// TIA Portal project "Modbus TCP Example with ESP32" (V16)

(* hardware
DEVICE "S7-1200 station_1"  S7-1200 Station
   slot 0: "Rack_0"  S7-1200 Rack  Rack  V1.0
   slot 1: "PLC_1"  CPU 1211C DC/DC/DC  6ES7 211-1AE40-0XB0  V4.4
*)

// ===== PLC "PLC_1"  CPU 1211C DC/DC/DC =====

VAR_GLOBAL   // PLC tag table "Default tag table"
   "Tag_1" AT %Q0.0 : Bool;
   "System_Byte" AT %MB1 : Byte;
   "FirstScan" AT %M1.0 : Bool;
   "DiagStatusUpdate" AT %M1.1 : Bool;
   "AlwaysTRUE" AT %M1.2 : Bool;
   "AlwaysFALSE" AT %M1.3 : Bool;
   "Clock_Byte" AT %MB0 : Byte;
   "Clock_10Hz" AT %M0.0 : Bool;
   "Clock_5Hz" AT %M0.1 : Bool;
   "Clock_2.5Hz" AT %M0.2 : Bool;
   "Clock_2Hz" AT %M0.3 : Bool;
   "Clock_1.25Hz" AT %M0.4 : Bool;
   "Clock_1Hz" AT %M0.5 : Bool;
   "Clock_0.625Hz" AT %M0.6 : Bool;
   "Clock_0.5Hz" AT %M0.7 : Bool;
END_VAR

TYPE "Modbus TCP FC01-02"
   STRUCT
      REQ : Bool := false;
      DISCONNECT : Bool := false;
      MODE : USInt;
      DATA_ADDR : UDInt;
      DATA_LEN : UInt := 40;
      CONNECT : TCON_IP_v4;
      DONE : Bool := false;
      BUSY : Bool := false;
      ERROR : Bool := false;
      STATUS : Word := 16#0;
      Data : Array[0..39] of Bool;
   END_STRUCT;
   // CONNECT.InterfaceId := 64;
   // CONNECT.ID := 1;
   // CONNECT.ConnectionType := 11;
   // CONNECT.ActiveEstablished := true;
   // CONNECT.RemoteAddress.ADDR[1] := 192;
   // CONNECT.RemoteAddress.ADDR[2] := 168;
   // CONNECT.RemoteAddress.ADDR[3] := 100;
   // CONNECT.RemoteAddress.ADDR[4] := 36;
   // CONNECT.RemotePort := 502;
END_TYPE

TYPE "Modbus TCP FC03-04"
   STRUCT
      REQ : Bool := false;
      DISCONNECT : Bool := false;
      MODE : USInt;
      DATA_ADDR : UDInt;
      DATA_LEN : UInt := 40;
      CONNECT : TCON_IP_v4;
      DONE : Bool := false;
      BUSY : Bool := false;
      ERROR : Bool := false;
      STATUS : Word := 16#0;
      Data : Array[0..39] of UInt;
   END_STRUCT;
   // CONNECT.InterfaceId := 64;
   // CONNECT.ID := 1;
   // CONNECT.ConnectionType := 11;
   // CONNECT.ActiveEstablished := true;
   // CONNECT.RemoteAddress.ADDR[1] := 192;
   // CONNECT.RemoteAddress.ADDR[2] := 168;
   // CONNECT.RemoteAddress.ADDR[3] := 100;
   // CONNECT.RemoteAddress.ADDR[4] := 36;
   // CONNECT.RemotePort := 502;
END_TYPE

DATA_BLOCK "Modbus client"   // DB3
{ S7_Optimized_Access := 'TRUE' }
VERSION : 0.1
   VAR
      Coils : "Modbus TCP FC01-02";
      "Discrete Inputs" : "Modbus TCP FC01-02";
      "Holding Registers" : "Modbus TCP FC03-04";
      "Input Registers" : "Modbus TCP FC03-04";
   END_VAR
BEGIN
   Coils.MODE := 1;
   Coils.DATA_ADDR := 1;
   "Discrete Inputs".MODE := 0;
   "Discrete Inputs".DATA_ADDR := 10101;
   "Discrete Inputs".DATA_LEN := 40;
   Coils.DATA_LEN := 40;
   "Holding Registers".MODE := 1;
   "Holding Registers".DATA_ADDR := 40201;
   "Holding Registers".DATA_LEN := 40;
   "Input Registers".MODE := 0;
   "Input Registers".DATA_ADDR := 30301;
   "Input Registers".DATA_LEN := 40;
END_DATA_BLOCK

ORGANIZATION_BLOCK "Main"   // OB1, LAD, ProgramCycle
TITLE = "Main Program Sweep (Cycle)"
{ S7_Optimized_Access := 'TRUE' }
VERSION : 0.1
   VAR_INPUT
      Initial_Call : Bool;   // Initial call of this OB
      Remanence : Bool;   // =True, if remanent data are available
   END_VAR
   VAR_TEMP
      start : Bool;
      trig1 : Bool;
      trig2 : Bool;
   END_VAR
BEGIN

REGION Network 1: Coils
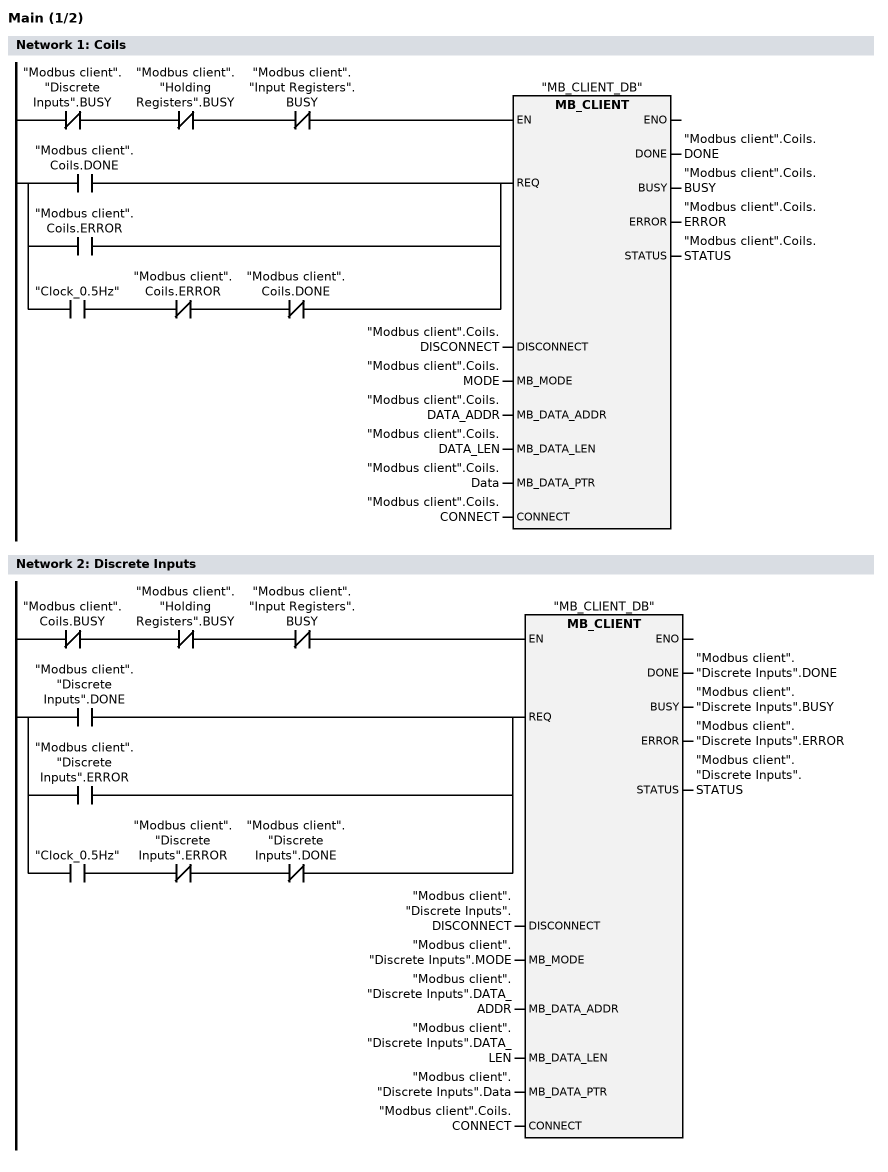
   IF NOT "Modbus client"."Discrete Inputs".BUSY AND NOT "Modbus client"."Holding Registers".BUSY AND NOT "Modbus client"."Input Registers".BUSY THEN
       "MB_CLIENT_DB"(REQ := "Modbus client".Coils.DONE OR "Modbus client".Coils.ERROR OR ("Clock_0.5Hz" AND NOT "Modbus client".Coils.ERROR AND NOT "Modbus client".Coils.DONE),   // MB_CLIENT
                      DISCONNECT := "Modbus client".Coils.DISCONNECT,
                      MB_MODE := "Modbus client".Coils.MODE,
                      MB_DATA_ADDR := "Modbus client".Coils.DATA_ADDR,
                      MB_DATA_LEN := "Modbus client".Coils.DATA_LEN,
                      MB_DATA_PTR := "Modbus client".Coils.Data,
                      CONNECT := "Modbus client".Coils.CONNECT,
                      DONE => "Modbus client".Coils.DONE,
                      BUSY => "Modbus client".Coils.BUSY,
                      ERROR => "Modbus client".Coils.ERROR,
                      STATUS => "Modbus client".Coils.STATUS);
   END_IF;
END_REGION

REGION Network 2: Discrete Inputs
   IF NOT "Modbus client".Coils.BUSY AND NOT "Modbus client"."Holding Registers".BUSY AND NOT "Modbus client"."Input Registers".BUSY THEN
       "MB_CLIENT_DB"(REQ := "Modbus client"."Discrete Inputs".DONE OR "Modbus client"."Discrete Inputs".ERROR OR ("Clock_0.5Hz" AND NOT "Modbus client"."Discrete Inputs".ERROR AND NOT "Modbus client"."Discrete Inputs".DONE),   // MB_CLIENT
                      DISCONNECT := "Modbus client"."Discrete Inputs".DISCONNECT,
                      MB_MODE := "Modbus client"."Discrete Inputs".MODE,
                      MB_DATA_ADDR := "Modbus client"."Discrete Inputs".DATA_ADDR,
                      MB_DATA_LEN := "Modbus client"."Discrete Inputs".DATA_LEN,
                      MB_DATA_PTR := "Modbus client"."Discrete Inputs".Data,
                      CONNECT := "Modbus client".Coils.CONNECT,
                      DONE => "Modbus client"."Discrete Inputs".DONE,
                      BUSY => "Modbus client"."Discrete Inputs".BUSY,
                      ERROR => "Modbus client"."Discrete Inputs".ERROR,
                      STATUS => "Modbus client"."Discrete Inputs".STATUS);
   END_IF;
END_REGION

REGION Network 3: Holding Registers
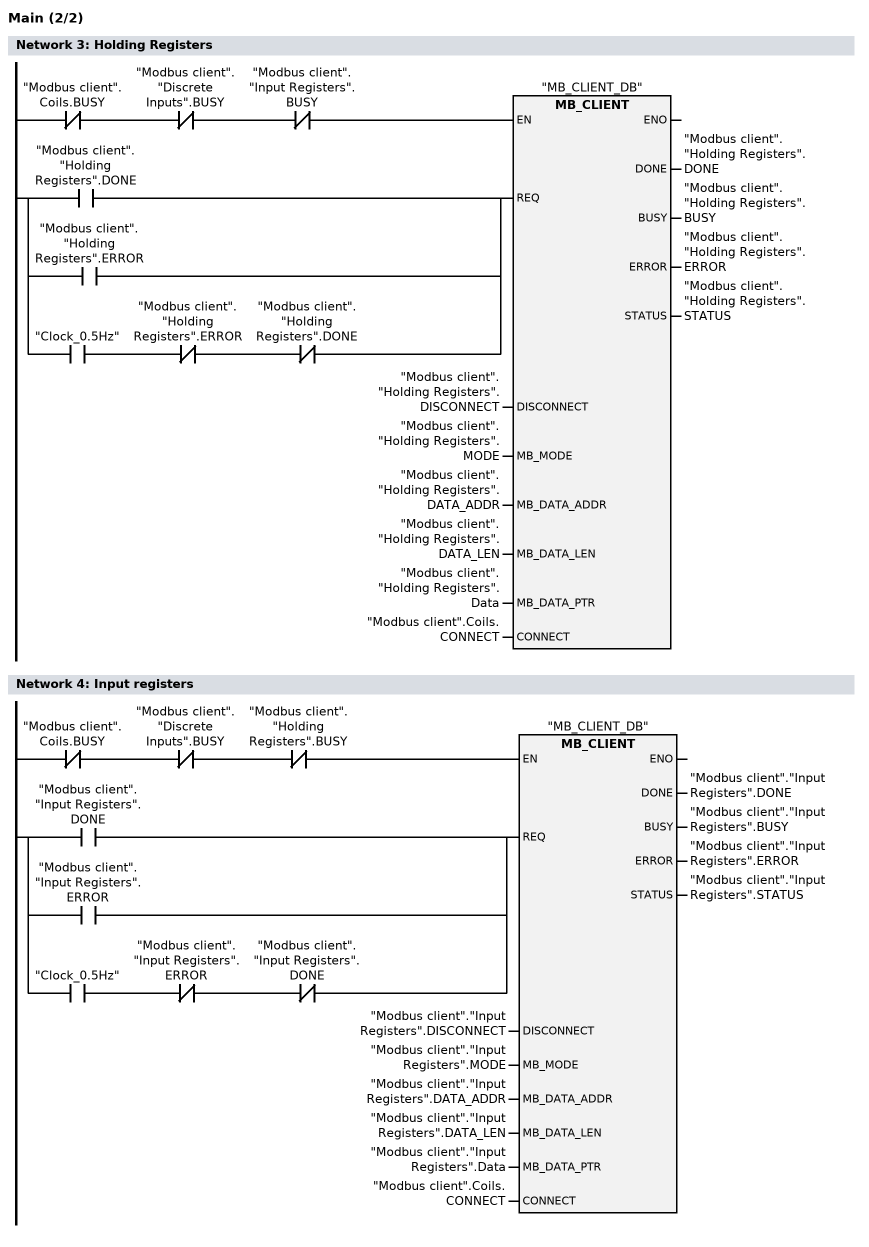
   IF NOT "Modbus client".Coils.BUSY AND NOT "Modbus client"."Discrete Inputs".BUSY AND NOT "Modbus client"."Input Registers".BUSY THEN
       "MB_CLIENT_DB"(REQ := "Modbus client"."Holding Registers".DONE OR "Modbus client"."Holding Registers".ERROR OR ("Clock_0.5Hz" AND NOT "Modbus client"."Holding Registers".ERROR AND NOT "Modbus client"."Holding Registers".DONE),   // MB_CLIENT
                      DISCONNECT := "Modbus client"."Holding Registers".DISCONNECT,
                      MB_MODE := "Modbus client"."Holding Registers".MODE,
                      MB_DATA_ADDR := "Modbus client"."Holding Registers".DATA_ADDR,
                      MB_DATA_LEN := "Modbus client"."Holding Registers".DATA_LEN,
                      MB_DATA_PTR := "Modbus client"."Holding Registers".Data,
                      CONNECT := "Modbus client".Coils.CONNECT,
                      DONE => "Modbus client"."Holding Registers".DONE,
                      BUSY => "Modbus client"."Holding Registers".BUSY,
                      ERROR => "Modbus client"."Holding Registers".ERROR,
                      STATUS => "Modbus client"."Holding Registers".STATUS);
   END_IF;
END_REGION

REGION Network 4: Input registers
   IF NOT "Modbus client".Coils.BUSY AND NOT "Modbus client"."Discrete Inputs".BUSY AND NOT "Modbus client"."Holding Registers".BUSY THEN
       "MB_CLIENT_DB"(REQ := "Modbus client"."Input Registers".DONE OR "Modbus client"."Input Registers".ERROR OR ("Clock_0.5Hz" AND NOT "Modbus client"."Input Registers".ERROR AND NOT "Modbus client"."Input Registers".DONE),   // MB_CLIENT
                      DISCONNECT := "Modbus client"."Input Registers".DISCONNECT,
                      MB_MODE := "Modbus client"."Input Registers".MODE,
                      MB_DATA_ADDR := "Modbus client"."Input Registers".DATA_ADDR,
                      MB_DATA_LEN := "Modbus client"."Input Registers".DATA_LEN,
                      MB_DATA_PTR := "Modbus client"."Input Registers".Data,
                      CONNECT := "Modbus client".Coils.CONNECT,
                      DONE => "Modbus client"."Input Registers".DONE,
                      BUSY => "Modbus client"."Input Registers".BUSY,
                      ERROR => "Modbus client"."Input Registers".ERROR,
                      STATUS => "Modbus client"."Input Registers".STATUS);
   END_IF;
END_REGION
END_ORGANIZATION_BLOCK